// TIA Portal V17 export
// export: Created 2023-12-22T15:28:36.2276932Z, ExportSetting WithDefaults, DisplayName Totally Integrated Automation Portal, DisplayVersion V17, DisplayName TIA Portal Openness, DisplayVersion V17, DisplayName TIA Portal Version Control Interface, DisplayVersion V17, DisplayName STEP 7 Professional, DisplayVersion V17, DisplayName STEP 7 Safety, DisplayVersion V17, DisplayName WinCC Advanced, DisplayVersion V17
DATA_BLOCK "V_D2_example_DB"   // DB700
VERSION : 0.1
// stored: AutoNumber false, DBAccessibleFromOPCUA true, InstanceOfName DRV_V_D2, InstanceOfType FB
"DRV_V_D2"
   // VAR_INPUT
   //    All_Block : Bool;
   // END_VAR
   // VAR_IN_OUT
   //    FB_QF : Bool;
   //    FB_KM_Open : Bool;
   //    FB_KM_Close : Bool;
   //    FB_Open : Bool;
   //    FB_Close : Bool;
   //    S_Alarm : Bool;
   //    CMD_Open : Bool;
   //    CMD_Close : Bool;
   // END_VAR
   // VAR RETAIN
   //    CMD : "CMD";
   //    Mode : Int;
   //    Status : Int;
   //    Use : Struct
   //       QF { S7_SetPoint := 'True'} : Bool;
   //       KM_Open { S7_SetPoint := 'True'} : Bool;
   //       KM_Close { S7_SetPoint := 'True'} : Bool;
   //       Open { S7_SetPoint := 'True'} : Bool;
   //       Close { S7_SetPoint := 'True'} : Bool;
   //       One_KM { S7_SetPoint := 'True'} : Bool;
   //       Electro { S7_SetPoint := 'True'} : Bool;
   //       Cross { S7_SetPoint := 'True'} : Bool;
   //       CMD_Open { S7_SetPoint := 'True'} : Bool;
   //       CMD_Close { S7_SetPoint := 'True'} : Bool;
   //       CMD_Reset : Bool;
   //       Local_Keys { S7_SetPoint := 'True'} : Bool;
   //       Local_EndPoint : Bool;
   //    END_STRUCT;
   //    FB : Struct
   //       QF : Bool;
   //       KM_Open : Bool;
   //       KM_Close : Bool;
   //       Open : Bool;
   //       Close : Bool;
   //       Reserv : Bool;
   //       Local_Open : Bool;
   //       Local_Close : Bool;
   //    END_STRUCT;
   //    ON : Bool;
   //    OFF : Bool;
   //    REQ_Open : Bool;
   //    REQ_Close : Bool;
   //    Tx { S7_SetPoint := 'True'} : Array[0..4] of "Time_S";
   //    Inv : Struct
   //       CMD { S7_SetPoint := 'True'} : Bool;
   //       QF { S7_SetPoint := 'True'} : Bool;
   //       KM_Open { S7_SetPoint := 'True'} : Bool;
   //       KM_Close { S7_SetPoint := 'True'} : Bool;
   //       Serivce { S7_SetPoint := 'True'} : Bool;
   //       Open { S7_SetPoint := 'True'} : Bool;
   //       Close { S7_SetPoint := 'True'} : Bool;
   //       Local_Open { S7_SetPoint := 'True'} : Bool;
   //       Local_Close { S7_SetPoint := 'True'} : Bool;
   //    END_STRUCT;
   //    Alarm : Struct
   //       Block : Bool;
   //       QF : Bool;
   //       KM_Open : Bool;
   //       KM_Close : Bool;
   //       Two_S : Bool;
   //       Open : Bool;
   //       Close : Bool;
   //       OpTime : Bool;
   //    END_STRUCT;
   //    Alarms : Word;
   //    Events : Word;
   //    pos : Array[0..15] of Bool;
   //    OpTime_h : DInt;
   //    OpTime_s { S7_SetPoint := 'True'} : DInt;
   //    CodeID { S7_SetPoint := 'True'} : Int;
   //    Indirect : Struct
   //       FB_QF { S7_SetPoint := 'True'} : Bool;
   //       FB_KM_Open { S7_SetPoint := 'True'} : Bool;
   //       FB_KM_Close { S7_SetPoint := 'True'} : Bool;
   //       FB_Open { S7_SetPoint := 'True'} : Bool;
   //       FB_Close { S7_SetPoint := 'True'} : Bool;
   //       CMD_Open { S7_SetPoint := 'True'} : Bool;
   //       CMD_Close { S7_SetPoint := 'True'} : Bool;
   //    END_STRUCT;
   //    Indirect_BYTE : Struct
   //       FB_QF { S7_SetPoint := 'True'} : Int;
   //       FB_KM_Open { S7_SetPoint := 'True'} : Int;
   //       FB_KM_Close { S7_SetPoint := 'True'} : Int;
   //       FB_Open { S7_SetPoint := 'True'} : Int;
   //       FB_Close { S7_SetPoint := 'True'} : Int;
   //       CMD_Open { S7_SetPoint := 'True'} : Int;
   //       CMD_Close { S7_SetPoint := 'True'} : Int;
   //       CMD_Reset : Int;
   //    END_STRUCT;
   //    Indirect_BIT : Struct
   //       FB_QF { S7_SetPoint := 'True'} : Int;
   //       FB_KM_Open { S7_SetPoint := 'True'} : Int;
   //       FB_KM_Close { S7_SetPoint := 'True'} : Int;
   //       FB_Open { S7_SetPoint := 'True'} : Int;
   //       FB_Close { S7_SetPoint := 'True'} : Int;
   //       CMD_Open { S7_SetPoint := 'True'} : Int;
   //       CMD_Close { S7_SetPoint := 'True'} : Int;
   //       CMD_Reset : Int;
   //    END_STRUCT;
   // END_VAR
BEGIN
END_DATA_BLOCK
